ABB RAPID module: MainModule.MOD

MODULE MainModule
	CONST robtarget home:=[[-11.36,-308.72,564.43],[0.00457441,-0.0108449,-0.999453,0.0309205],[-2,-1,-2,0],[9E+09,9E+09,9E+09,9E+09,9E+09,9E+09]];
	CONST robtarget qld:=[[-137.82,-448.70,310.91],[0.00456574,-0.0108441,-0.999453,0.0309185],[-2,0,-2,0],[9E+09,9E+09,9E+09,9E+09,9E+09,9E+09]];
	CONST robtarget mdd{3,2}:=[[[[361.60,-54.76,372.99],[0.0194415,0.713713,0.699732,0.0247066],[-1,0,0,0],[9E+09,9E+09,9E+09,9E+09,9E+09,9E+09]],[[400.63,-52.09,374.66],[0.0193602,0.713759,0.699689,0.0246723],[-1,0,0,0],[9E+09,9E+09,9E+09,9E+09,9E+09,9E+09]]],[[[358.90,13.35,373.52],[0.0193917,0.713731,0.699715,0.0247161],[0,0,1,0],[9E+09,9E+09,9E+09,9E+09,9E+09,9E+09]],[[399.43,17.06,377.41],[0.0193733,0.713742,0.699706,0.0246732],[0,0,1,0],[9E+09,9E+09,9E+09,9E+09,9E+09,9E+09]]],[[[356.49,83.11,374.28],[0.0194372,0.71373,0.699715,0.0247205],[0,-1,1,0],[9E+09,9E+09,9E+09,9E+09,9E+09,9E+09]],[[397.18,83.44,373.21],[0.0194051,0.713751,0.699695,0.0247007],[0,-1,1,0],[9E+09,9E+09,9E+09,9E+09,9E+09,9E+09]]]];
	PROC main()
		<SMT>
	ENDPROC
ENDMODULE
